{attribute 'qualified_only'}
VAR_GLOBAL
	// Simulation on for whole project
	g_bCmdSimulationOn	: BOOL;
END_VAR

(* stored: Version 1.1.0.1, ProductVersion 3.1.4024.10
   GVL GVL: Id {ca8c3cb0-b92b-4ea5-9dfc-8c13386c714b} *)
